PROGRAM P_Demo_FB_DMXSetLampOnMode
VAR
    fbSetLampOnMode   : FB_DMXSetLampOnMode;          // 写开灯模式
    stDmxCmdBuffer    : ST_DMXCommandBuffer;          // 与通讯 FB 共用
    wTargetManufId    : WORD := 16#4241;              // 目标灯具厂商 ID
    dwTargetDeviceId  : DWORD := 16#12131415;         // 目标灯具设备 ID
    byTargetPort      : BYTE := 0;                    // 根设备通道 0
    eNewOnMode        : E_DMXLampOnMode := eDMXLampOnModeDMX;  // 仅收到 DMX 数据时点亮
    bDoSet            : BOOL := FALSE;                // 在线给一次上升沿触发
    bBusy             : BOOL;
    bError            : BOOL;
    udiErrId          : UDINT;
END_VAR

// ============================================================
// Tc2_DMX.FB_DMXSetLampOnMode 演示程序
// ============================================================
// 场景：批量配置新装灯具上电行为，统一设为收到 DMX 数据后才点亮，避免上电满亮刺眼。
// 价值：把开灯策略下发做成 PLC 调用，可对全场灯具批量统一配置，无需逐台进本地菜单。
// 验证：设 eNewOnMode，给 bDoSet 一次上升沿 -> bBusy 短暂 TRUE -> 回 FALSE 后用 FB_DMXGetLampOnMode 回读应等于所设值。
// 验证步骤：
//   1. 右键 PLC 项目下 POUs 文件夹 → Add → Existing Item → 选本 .TcPOU 文件
//   2. 引用 Tc2_DMX；同项目里放一个 FB_EL6851CommunicationEx 实例并共用 stDmxCmdBuffer（非 CycleMode）
//   3. 编译 → 登录 → 运行；按上方『验证』行在线给上升沿观察
// ============================================================

fbSetLampOnMode(
    bStart                     := bDoSet,
    wDestinationManufacturerId := wTargetManufId,
    dwDestinationDeviceId      := dwTargetDeviceId,
    byPortId                   := byTargetPort,
    eLampOnMode                := eNewOnMode,
    dwOptions                  := 0,
    stCommandBuffer            := stDmxCmdBuffer,
    bBusy                      => bBusy,
    bError                     => bError,
    udiErrorId                 => udiErrId
);

END_PROGRAM

(* stored: Version 1.1.0.1, ProductVersion 3.1.4024.5
   POU P_Demo_FB_DMXSetLampOnMode: Id {352f29eb-5177-57c1-8399-c113518aad30}, SpecialFunc None *)
